Universal Robots PolyScope program: test_calibration.urp

Program test_calibration (installation=default directory=/programs/HandEyeCalibration createdIn=5.9.1.1031110 lastSavedIn=5.9.1.1031110 robotSerialNumber=20185500256)
Calibrated DH parameters: a=[0.000163, -0.146131, -0.38577, 0.000126, -0.000021, 0]; d=[0.161954, 188.306531, -157.478086, -30.695088, 0.099716, 0.099628]; alpha=[1.569701, -0.00212, 0.002263, 1.570438, -1.570123, 0]; deltaTheta=[0, -1.219859, 7.681919, -0.178877, -0.000001, 0]
Robot Program (runOnlyOnce=true)
  MoveJ speed 60 deg/s, acceleration 80 deg/s^2 (useActiveTCP=false) tcp=TCP_calib_stick; feature=Base
    Waypoint Waypoint_1: TCP in base x=-2.828 y=-210.201 z=305.114 mm, rx=1.391 ry=1.1781 rz=1.091 rad; joints [89.744, -126.495, 122.598, -82.858, -96.348, 97.161] deg; TCP offset x=1.48 y=-110.3 z=134.52 mm, rx=-1.567 ry=0 rz=0 rad
  Set NoAction tcp=TCP_cam
  board_pose := p_rel(get_actual_tcp_pose(),p[0.0175,-0.2235,0.42188,0,0,0])
  board_pose := p_rel(board_pose,p[0,0,0,3.14,0,0])
  Script: board_pose[2] = board_pose[2]+0.01
  SuppressedNode
    MoveJ speed 60 deg/s, acceleration 80 deg/s^2 (useActiveTCP=true) feature=Base
      Waypoint Waypoint_2: TCP in base x=-38.451 y=-419.47 z=319.723 mm, rx=1.7719 ry=0.3448 rz=1.3719 rad; joints [51.329, -90.858, 105.717, -22.65, -12.248, 138.308] deg; TCP offset x=-56.7 y=32.5 z=6.2 mm, rx=-0.0037 ry=-0.0098 rz=-1.5604 rad
  Set NoAction tcp=TCP_calib_stick
  MoveL speed 250 mm/s, acceleration 1200 mm/s^2 (useActiveTCP=true) feature=Base
    Waypoint Waypoint (Variable): variable(name=board_pose)
